// FB_HekBesturing.scl
// Toestandsmachine voor hekbesturing - 9 toestanden per FDS sectie 2.2
// Hoofdlogica voor automatisch hek met veiligheidsprioriteiten
//
// Toestanden (per DB_States):
// 0 = HOMING      - Zoeken referentiepositie bij opstart
// 1 = IDLE_OPEN   - Hek volledig open, motor uit
// 2 = IDLE_DICHT  - Hek volledig dicht, alarm aan
// 3 = MOVING_OPEN - Beweging richting open
// 4 = MOVING_DICHT- Beweging richting dicht
// 5 = STOPPED     - Gestopt in tussenpositie
// 6 = VS_PAUSE    - Gepauzeerd door lichtsluis
// 7 = PBV_RETRACT - Terugtrekken na bumperactivatie
// 8 = FAULT       - Sensorstoring gedetecteerd

FUNCTION_BLOCK "FB_HekBesturing"
{ S7_Optimized_Access := 'TRUE' }
VERSION : 0.1

   VAR_INPUT
      i_SS_Open : Bool;              // Sleutelschakelaar naar OPEN (1=contact)
      i_SS_Dicht : Bool;             // Sleutelschakelaar naar DICHT (1=contact)
      i_DK_Bediening : Bool;         // Drukknop bediening (NC: 0=ingedrukt)
      i_BNS_Open : Bool;             // Benaderingsschakelaar OPEN (NC: 0=bereikt)
      i_BNS_Dicht : Bool;            // Benaderingsschakelaar DICHT (NC: 0=bereikt)
      i_PBV_Trigger : Bool;          // PBV actief (van FC_Veiligheid)
      i_VS_Trigger : Bool;           // VS actief (van FC_Veiligheid)
      i_Fault : Bool;                // Sensordefect (van FC_Veiligheid)
   END_VAR

   VAR_OUTPUT
      q_MS_Open : Bool;              // Motor sturing richting OPEN
      q_MS_Dicht : Bool;             // Motor sturing richting DICHT
      q_MS_LaagToeren : Bool;        // Motor lage snelheid actief
      q_AlarmKerk : Bool;            // Kerkalarm (0=hek dicht, 1=hek niet dicht)
      q_HuidigeToestand : Int;       // Huidige toestand voor diagnose/HMI
   END_VAR

   VAR
      m_Toestand : Int;              // Huidige toestand van de state machine
      m_VorigeToestand : Int;        // Vorige toestand (voor transitie detectie)
      m_LaatsteRichting : Int;       // Laatst actieve richting (DIR_OPEN=1, DIR_DICHT=2)
      m_VorigeRichtingVoorVS : Int;  // Direction before VS pause (for auto-resume)

      // Edge detection - IEC standard function blocks
      m_EdgeSS_Open : R_TRIG;        // Rising edge key switch OPEN
      m_EdgeSS_Dicht : R_TRIG;       // Rising edge key switch DICHT
      m_EdgeDK : F_TRIG;             // Falling edge push button (NC: 0=pressed)

      // Timers - existing
      m_TON_Timeout : TON;           // Movement timeout (90s per CFG_BewegingTimeoutS)
      m_TON_PBV_Retract : TON;       // PBV retract duration timer (3s per CFG_PBV_TerugtrekMs)

      // Timers - TONR for pausable low speed (TMR-08)
      m_TONR_LaagToeren : TONR;      // Normal start low speed (5s)
      m_TONR_VS_LaagToeren : TONR;   // Post-VS resume low speed (2s)

      // Timers - TON for fixed delays
      m_TON_VS_Hervatting : TON;     // VS resume delay (2s)
      m_TON_PBV_Pauze : TON;         // PBV pause before retract (500ms)

      // Direction change tracking (TMR-08: reset on direction change)
      m_VorigeRichting : Int;        // Previous direction for change detection

      // Timer output captures (captured once per scan per TMR-09)
      m_LowSpeedDone : Bool;         // Start low speed timer complete
      m_VS_LowSpeedDone : Bool;      // VS low speed timer complete
      m_VS_ResumeDelayDone : Bool;   // VS resume delay complete
      m_PBV_PauseDone : Bool;        // PBV pause complete

      // State tracking flags
      m_VS_ResumeActive : Bool;      // Flag: currently resuming from VS (for VS low speed)
      m_PBV_Retracting : Bool;       // Flag: PBV retract in progress (after pause)

      // Control flags
      m_KeyReleased : Bool := TRUE;  // CTL-08: Key release tracking after timeout
      m_FirstScan : Bool := TRUE;    // Power-on detection for initialization
   END_VAR

VAR_TEMP
    t_DirectionChanged : Bool;     // Direction change detected this scan
    t_MotorMoving : Bool;          // Motor in normal movement state
    t_ReachedEndstop : Bool;       // At endstop (for timer reset)
    t_InMovement : Bool;           // In any movement state (for low speed calc)
    t_NormalLowSpeed : Bool;       // Normal start low speed needed
    t_VS_LowSpeed : Bool;          // VS resume low speed needed
END_VAR

BEGIN
    // =========================================================================
    // Edge detection - call BEFORE CASE statement (ensures edges detected once per scan)
    // =========================================================================
    #m_EdgeSS_Open(CLK := #i_SS_Open);
    #m_EdgeSS_Dicht(CLK := #i_SS_Dicht);
    #m_EdgeDK(CLK := #i_DK_Bediening);  // NC: falling edge = press

    // =========================================================================
    // Movement timeout timer - runs in HOMING, MOVING_OPEN, MOVING_DICHT
    // =========================================================================
    #m_TON_Timeout(IN := (#m_Toestand = "DB_States".STATE_HOMING) OR
                          (#m_Toestand = "DB_States".STATE_MOVING_OPEN) OR
                          (#m_Toestand = "DB_States".STATE_MOVING_DICHT),
                   PT := "DB_Config".Timers.CFG_BewegingTimeoutS);

    // =========================================================================
    // PBV retract timer - runs only during retract phase (after pause)
    // =========================================================================
    #m_TON_PBV_Retract(IN := (#m_Toestand = "DB_States".STATE_PBV_RETRACT) AND #m_PBV_Retracting,
                       PT := "DB_Config".Timers.CFG_PBV_TerugtrekMs);

    // =========================================================================
    // Direction change detection (TMR-08: reset timer on direction change)
    // =========================================================================
    #t_DirectionChanged := (#m_LaatsteRichting <> #m_VorigeRichting) AND
                           (#m_LaatsteRichting <> "DB_States".DIR_NONE) AND
                           (#m_VorigeRichting <> "DB_States".DIR_NONE);
    #m_VorigeRichting := #m_LaatsteRichting;

    // =========================================================================
    // Computed conditions for timer logic
    // =========================================================================
    // Motor moving in normal movement states
    #t_MotorMoving := (#m_Toestand = "DB_States".STATE_MOVING_OPEN) OR
                      (#m_Toestand = "DB_States".STATE_MOVING_DICHT);

    // Reached endstop (timer reset condition) - NC: 0 = reached
    #t_ReachedEndstop := (NOT #i_BNS_Open) OR (NOT #i_BNS_Dicht);

    // =========================================================================
    // Low speed timer - pausable TONR (TMR-01, TMR-08)
    // Accumulates during movement, pauses on stop, resets on direction change
    // =========================================================================
    #m_TONR_LaagToeren(
        IN := #t_MotorMoving,
        PT := "DB_Config".Timers.CFG_LaagToerenMs,
        R := #t_DirectionChanged OR #t_ReachedEndstop,
        Q => #m_LowSpeedDone
    );

    // =========================================================================
    // Post-VS resume low speed timer (TMR-05)
    // =========================================================================
    #m_TONR_VS_LaagToeren(
        IN := #t_MotorMoving AND #m_VS_ResumeActive,
        PT := "DB_Config".Timers.CFG_VS_LaagToerenMs,
        R := #t_DirectionChanged OR #t_ReachedEndstop OR (NOT #m_VS_ResumeActive),
        Q => #m_VS_LowSpeedDone
    );

    // =========================================================================
    // VS resume delay timer (TMR-04)
    // =========================================================================
    #m_TON_VS_Hervatting(
        IN := (#m_Toestand = "DB_States".STATE_VS_PAUSE) AND (NOT #i_VS_Trigger),
        PT := "DB_Config".Timers.CFG_VS_HervattingMs,
        Q => #m_VS_ResumeDelayDone
    );

    // =========================================================================
    // PBV pause timer (TMR-02)
    // =========================================================================
    #m_TON_PBV_Pauze(
        IN := (#m_Toestand = "DB_States".STATE_PBV_RETRACT) AND (NOT #m_PBV_Retracting),
        PT := "DB_Config".Timers.CFG_PBV_PauzeMs,
        Q => #m_PBV_PauseDone
    );

    // =========================================================================
    // Power-on initialization - determine initial state from endstops
    // =========================================================================
    IF #m_FirstScan THEN
        #m_FirstScan := FALSE;
        // NC sensors: 0 = reached, 1 = not reached
        IF (NOT #i_BNS_Open) AND (NOT #i_BNS_Dicht) THEN
            // Both endstops - sensor fault
            #m_Toestand := "DB_States".STATE_FAULT;
        ELSIF NOT #i_BNS_Dicht THEN
            // At DICHT position
            #m_Toestand := "DB_States".STATE_IDLE_DICHT;
        ELSIF NOT #i_BNS_Open THEN
            // At OPEN position
            #m_Toestand := "DB_States".STATE_IDLE_OPEN;
        ELSE
            // Neither endstop - unknown position, need homing
            #m_Toestand := "DB_States".STATE_HOMING;
        END_IF;
    END_IF;

    // =========================================================================
    // Save previous state (for transition detection in future plans)
    // =========================================================================
    #m_VorigeToestand := #m_Toestand;

    // =========================================================================
    // Main state machine CASE statement
    // =========================================================================
    CASE #m_Toestand OF
        "DB_States".STATE_HOMING:
            // HOMING: Moving toward DICHT to find reference position
            // Safety checks FIRST (priority: FAULT > PBV > VS per CONTEXT.md)
            IF #i_Fault THEN
                #m_Toestand := "DB_States".STATE_FAULT;
            ELSIF #i_PBV_Trigger OR #i_VS_Trigger THEN
                // SM-04: HOMING aborts to STOPPED on PBV or VS trigger
                #m_Toestand := "DB_States".STATE_STOPPED;
            ELSIF #m_TON_Timeout.Q THEN
                // SAF-12: HOMING uses same timeout as normal movement
                #m_Toestand := "DB_States".STATE_STOPPED;
                #m_KeyReleased := FALSE;
            ELSIF NOT #i_BNS_Dicht THEN
                // NC: 0 = reached DICHT endstop
                #m_Toestand := "DB_States".STATE_IDLE_DICHT;
            ELSIF #m_EdgeDK.Q THEN
                // Push button during HOMING -> abort to STOPPED (manual stop works in all movement states)
                #m_Toestand := "DB_States".STATE_STOPPED;
            END_IF;
            // Motor output: moving toward DICHT (handled in output section)

        "DB_States".STATE_IDLE_OPEN:
            // Gate fully OPEN, motor off
            // Clear direction memory when at endstop (no accidental resume toward wall)
            #m_LaatsteRichting := "DB_States".DIR_NONE;

            IF #i_Fault THEN
                #m_Toestand := "DB_States".STATE_FAULT;
            ELSIF #i_PBV_Trigger THEN
                // PBV at IDLE_OPEN: stay here (already at safest position per CONTEXT.md)
                ; // No action - already at OPEN endstop
            // Key DICHT starts movement toward DICHT
            ELSIF #m_EdgeSS_Dicht.Q THEN
                #m_Toestand := "DB_States".STATE_MOVING_DICHT;
                #m_LaatsteRichting := "DB_States".DIR_DICHT;
            END_IF;
            // No push button action from IDLE (no direction memory)

        "DB_States".STATE_IDLE_DICHT:
            // Gate fully CLOSED, motor off, alarm deactivated
            // Clear direction memory when at endstop
            #m_LaatsteRichting := "DB_States".DIR_NONE;

            IF #i_Fault THEN
                #m_Toestand := "DB_States".STATE_FAULT;
            // Key OPEN starts movement toward OPEN
            ELSIF #m_EdgeSS_Open.Q THEN
                #m_Toestand := "DB_States".STATE_MOVING_OPEN;
                #m_LaatsteRichting := "DB_States".DIR_OPEN;
            END_IF;
            // No push button action from IDLE (no direction memory)

        "DB_States".STATE_MOVING_OPEN:
            // Moving toward OPEN position
            // Safety checks FIRST (priority: FAULT > PBV > VS)
            IF #i_Fault THEN
                #m_Toestand := "DB_States".STATE_FAULT;
            ELSIF #i_PBV_Trigger THEN
                // PBV during OPEN movement -> retract (continues toward OPEN)
                #m_Toestand := "DB_States".STATE_PBV_RETRACT;
            ELSIF #i_VS_Trigger THEN
                // VS pause - save direction for auto-resume
                #m_VorigeRichtingVoorVS := "DB_States".DIR_OPEN;
                #m_Toestand := "DB_States".STATE_VS_PAUSE;
            ELSIF #m_TON_Timeout.Q THEN
                // SAF-11: Movement timeout -> STOPPED
                #m_Toestand := "DB_States".STATE_STOPPED;
                #m_KeyReleased := FALSE;  // CTL-08: require key release
            ELSIF NOT #i_BNS_Open THEN
                // NC: 0 = reached OPEN endstop
                #m_Toestand := "DB_States".STATE_IDLE_OPEN;
            ELSIF #m_EdgeDK.Q THEN
                // Push button -> manual stop
                #m_Toestand := "DB_States".STATE_STOPPED;
            ELSIF #m_EdgeSS_Dicht.Q THEN
                // CTL-07: Opposing key direction while moving -> stop
                #m_Toestand := "DB_States".STATE_STOPPED;
            END_IF;
            // Direction memory maintained (already set when entering this state)
            // Motor output: q_MS_Open=TRUE (handled in output section)

        "DB_States".STATE_MOVING_DICHT:
            // Moving toward DICHT (closed) position
            // Safety checks FIRST (priority: FAULT > PBV > VS)
            IF #i_Fault THEN
                #m_Toestand := "DB_States".STATE_FAULT;
            ELSIF #i_PBV_Trigger THEN
                // PBV during DICHT movement -> retract toward OPEN (SAF-03)
                #m_Toestand := "DB_States".STATE_PBV_RETRACT;
            ELSIF #i_VS_Trigger THEN
                // VS pause - save direction for auto-resume
                #m_VorigeRichtingVoorVS := "DB_States".DIR_DICHT;
                #m_Toestand := "DB_States".STATE_VS_PAUSE;
            ELSIF #m_TON_Timeout.Q THEN
                // SAF-11: Movement timeout -> STOPPED
                #m_Toestand := "DB_States".STATE_STOPPED;
                #m_KeyReleased := FALSE;  // CTL-08: require key release
            ELSIF NOT #i_BNS_Dicht THEN
                // NC: 0 = reached DICHT endstop
                #m_Toestand := "DB_States".STATE_IDLE_DICHT;
            ELSIF #m_EdgeDK.Q THEN
                // Push button -> manual stop
                #m_Toestand := "DB_States".STATE_STOPPED;
            ELSIF #m_EdgeSS_Open.Q THEN
                // CTL-07: Opposing key direction while moving -> stop
                #m_Toestand := "DB_States".STATE_STOPPED;
            END_IF;
            // Direction memory maintained (already set when entering this state)
            // Motor output: q_MS_Dicht=TRUE (handled in output section)

        "DB_States".STATE_STOPPED:
            // Stopped in intermediate position (not at endstop)
            // Motor outputs off (handled in output section)

            IF #i_Fault THEN
                #m_Toestand := "DB_States".STATE_FAULT;
            ELSE
                // CTL-08: Track key release after timeout
                // Keys must be released before new input is accepted
                IF NOT #m_KeyReleased THEN
                    // Waiting for key release after timeout
                    IF NOT #i_SS_Open AND NOT #i_SS_Dicht THEN
                        #m_KeyReleased := TRUE;
                    END_IF;
                    // Ignore all input while waiting for release
                ELSE
                    // Normal input processing
                    // CTL-06: Key switch from STOPPED starts in selected direction (overrides last direction)
                    IF #m_EdgeSS_Open.Q THEN
                        #m_Toestand := "DB_States".STATE_MOVING_OPEN;
                        #m_LaatsteRichting := "DB_States".DIR_OPEN;
                    ELSIF #m_EdgeSS_Dicht.Q THEN
                        #m_Toestand := "DB_States".STATE_MOVING_DICHT;
                        #m_LaatsteRichting := "DB_States".DIR_DICHT;
                    // CTL-04, CTL-05: Push button toggles stop/resume, resumes last direction
                    ELSIF #m_EdgeDK.Q THEN
                        IF #m_LaatsteRichting = "DB_States".DIR_OPEN THEN
                            #m_Toestand := "DB_States".STATE_MOVING_OPEN;
                        ELSIF #m_LaatsteRichting = "DB_States".DIR_DICHT THEN
                            #m_Toestand := "DB_States".STATE_MOVING_DICHT;
                        END_IF;
                        // If m_LaatsteRichting = DIR_NONE (fresh power-up, never moved)
                        // -> ignore push button (safest default per CONTEXT.md - no movement without explicit direction)
                    END_IF;
                END_IF;
            END_IF;

        "DB_States".STATE_VS_PAUSE:
            // Paused due to vehicle sensor (beam blocked)
            // SAF-08: Auto-resumes in same direction when beam clears
            // SAF-09: Ignores operator input during pause (auto-resume has priority)
            // Motor outputs OFF (handled in output section - not in MOVING states)

            // Safety checks FIRST (priority: FAULT > PBV > VS)
            IF #i_Fault THEN
                #m_Toestand := "DB_States".STATE_FAULT;
            ELSIF #i_PBV_Trigger THEN
                // PBV > VS: PBV can interrupt VS_PAUSE (statemachine.mmd line 49)
                #m_Toestand := "DB_States".STATE_PBV_RETRACT;
                #m_PBV_Retracting := FALSE;  // Start fresh - pause phase first
            ELSIF NOT #i_VS_Trigger THEN
                // Beam cleared - wait for resume delay (TMR-04)
                IF #m_VS_ResumeDelayDone THEN
                    // TMR-04 complete: resume movement with low speed
                    #m_VS_ResumeActive := TRUE;  // Flag for VS low speed timer
                    IF #m_VorigeRichtingVoorVS = "DB_States".DIR_OPEN THEN
                        #m_Toestand := "DB_States".STATE_MOVING_OPEN;
                    ELSIF #m_VorigeRichtingVoorVS = "DB_States".DIR_DICHT THEN
                        #m_Toestand := "DB_States".STATE_MOVING_DICHT;
                    ELSE
                        // Safety fallback: no saved direction -> go to STOPPED
                        #m_Toestand := "DB_States".STATE_STOPPED;
                    END_IF;
                END_IF;
                // Note: If beam re-triggers during delay, timer resets (TON behavior)
            END_IF;
            // NOTE: Push button and key switch edges are IGNORED in this state (SAF-09)
            // Auto-resume has priority over operator input

        "DB_States".STATE_PBV_RETRACT:
            // Retracting toward OPEN after bumper activation
            // SAF-03: Always moves toward OPEN regardless of previous direction
            // SAF-05: Ignores ALL operator input during retract
            // TMR-02: Wait CFG_PBV_PauzeMs before starting movement
            // TMR-03: Max retract duration CFG_PBV_TerugtrekMs

            // Only FAULT can interrupt PBV_RETRACT (FAULT > PBV priority)
            IF #i_Fault THEN
                #m_Toestand := "DB_States".STATE_FAULT;
                #m_PBV_Retracting := FALSE;  // Reset for next time
            ELSIF NOT #m_PBV_Retracting THEN
                // PAUSE PHASE: Waiting before retract (TMR-02)
                // m_TON_PBV_Pauze runs in timer section when in this state AND NOT m_PBV_Retracting
                IF #m_PBV_PauseDone THEN
                    // Pause complete - start retract movement
                    #m_PBV_Retracting := TRUE;
                END_IF;
                // Motor outputs are OFF during pause (handled in output section)
            ELSE
                // RETRACT PHASE: Moving toward OPEN (motor active)
                IF NOT #i_BNS_Open THEN
                    // NC: 0 = reached OPEN endstop -> safest position achieved
                    #m_Toestand := "DB_States".STATE_IDLE_OPEN;
                    #m_PBV_Retracting := FALSE;  // Reset for next time
                ELSIF #m_TON_PBV_Retract.Q THEN
                    // SAF-04: Max retract duration reached, still in mid-position
                    #m_Toestand := "DB_States".STATE_STOPPED;
                    #m_LaatsteRichting := "DB_States".DIR_NONE;  // Clear direction memory
                    #m_PBV_Retracting := FALSE;  // Reset for next time
                END_IF;
            END_IF;
            // NOTE: Push button and key switch edges are IGNORED in this state (SAF-05)
            // They are still detected (edge triggers run before CASE) but not acted upon

        "DB_States".STATE_FAULT:
            // Sensor fault detected - both endstops active simultaneously
            // Motor outputs forced off (handled in output section)
            // Clear direction memory on FAULT (safety per CONTEXT.md - Claude decides)
            #m_LaatsteRichting := "DB_States".DIR_NONE;

            // Auto-recovery when fault condition clears (SM-08)
            IF NOT #i_Fault THEN
                // Check current sensor state to determine recovery state
                IF NOT #i_BNS_Dicht THEN
                    #m_Toestand := "DB_States".STATE_IDLE_DICHT;
                ELSIF NOT #i_BNS_Open THEN
                    #m_Toestand := "DB_States".STATE_IDLE_OPEN;
                ELSE
                    // Neither endstop - go to STOPPED (safe default per CONTEXT.md)
                    #m_Toestand := "DB_States".STATE_STOPPED;
                END_IF;
            END_IF;

        ELSE
            // Unexpected state - recover to safe state
            #m_Toestand := "DB_States".STATE_STOPPED;
    END_CASE;

    // =========================================================================
    // Motor outputs based on state (direction only, low speed in Phase 4)
    // =========================================================================
    CASE #m_Toestand OF
        "DB_States".STATE_MOVING_OPEN:
            #q_MS_Open := TRUE;
            #q_MS_Dicht := FALSE;

        "DB_States".STATE_PBV_RETRACT:
            // Only output motor during retract phase (after pause)
            IF #m_PBV_Retracting THEN
                #q_MS_Open := TRUE;
                #q_MS_Dicht := FALSE;
            ELSE
                // Pause phase - motor off
                #q_MS_Open := FALSE;
                #q_MS_Dicht := FALSE;
            END_IF;

        "DB_States".STATE_MOVING_DICHT, "DB_States".STATE_HOMING:
            #q_MS_Open := FALSE;
            #q_MS_Dicht := TRUE;

        ELSE
            #q_MS_Open := FALSE;
            #q_MS_Dicht := FALSE;
    END_CASE;

    // =========================================================================
    // Low speed output determination (TMR-01, TMR-05)
    // =========================================================================
    // Low speed active when:
    // 1. In HOMING (always low speed per FDS 2.2)
    // 2. In PBV_RETRACT (always low speed per FDS 5.2)
    // 3. In MOVING_* and start timer not complete (first CFG_LaagToerenMs)
    // 4. In MOVING_* after VS resume and VS timer not complete (CFG_VS_LaagToerenMs)

    #t_InMovement := (#m_Toestand = "DB_States".STATE_MOVING_OPEN) OR
                     (#m_Toestand = "DB_States".STATE_MOVING_DICHT);

    // Normal start low speed: during movement, timer not complete
    #t_NormalLowSpeed := #t_InMovement AND NOT #m_LowSpeedDone;

    // VS resume low speed: after VS, timer not complete
    #t_VS_LowSpeed := #t_InMovement AND #m_VS_ResumeActive AND NOT #m_VS_LowSpeedDone;

    // Final low speed determination
    #q_MS_LaagToeren := (#m_Toestand = "DB_States".STATE_HOMING) OR
                        (#m_Toestand = "DB_States".STATE_PBV_RETRACT) OR
                        #t_NormalLowSpeed OR
                        #t_VS_LowSpeed;

    // Clear VS resume flag when VS low speed complete or at endstop
    IF #m_VS_LowSpeedDone OR #t_ReachedEndstop THEN
        #m_VS_ResumeActive := FALSE;
    END_IF;

    // Alarm: only deactivated (0) when in IDLE_DICHT
    #q_AlarmKerk := NOT (#m_Toestand = "DB_States".STATE_IDLE_DICHT);

    // Diagnostic output
    #q_HuidigeToestand := #m_Toestand;

END_FUNCTION_BLOCK
